(* Logix 5000 project; controller Lift_Station_Template vendor 1 type 14 code 196 rev 32.11; software revision 32.00 *)

TASK MainTask (continuous, watchdog 500 ms) : InLink, MainProgram, OutLink

MODULES
   Local : vendor 1 type 14 code 196 (5069 0, rev 32.11)
      DI_01 : 5069-IB16 (5069 1, rev 2.1, StandardDataDriven RPI 5 ms)
      DO_02 : 5069-OB16 (5069 2, rev 2.1, StandardDataDriven RPI 5 ms)
END_MODULES

TYPE Pump :
STRUCT
   HOA_Auto : BOOL;   // Physical HOA in Auto
   ManStartPB : BOOL;
   ManStopPB : BOOL;
   AutoStart : BOOL;
   CallToRun : BOOL;
   Running : BOOL;
   FailToRun : DiscreteAlarm;
   StartCount : DINT;
   ManSS : BOOL;
END_STRUCT
END_TYPE

ADD_ON_INSTRUCTION DiscreteAlarm   (* revision 1.0 *)
VAR_INPUT
   Trigger : BOOL; {required}
   Delay : DINT; {required}
   Supress : BOOL; {visible}
   Disable : BOOL; {visible}
END_VAR
VAR_OUTPUT
   Alarm : BOOL; {required}
   Acc : DINT; {visible}
END_VAR
VAR_INPUT
   Latching : BOOL; {visible}
   Reset : BOOL;
END_VAR
VAR
   DelayTmr : TIMER; {access None}
END_VAR

ROUTINE Logic   (* ladder *)
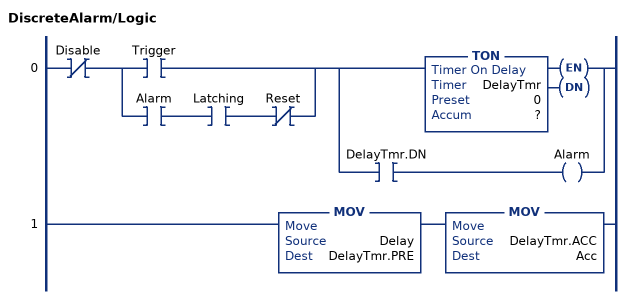
   0: XIO(Disable)[XIC(Trigger) ,XIC(Alarm) XIC(Latching) XIO(Reset) ][TON(DelayTmr,?,?) ,XIC(DelayTmr.DN) OTE(Alarm) ];
   1: MOV(Delay,DelayTmr.PRE)MOV(DelayTmr.ACC,Acc);
END_ROUTINE
END_ADD_ON_INSTRUCTION

VAR_GLOBAL   (* controller tags *)
   LSH_2 : BOOL;
   LSL_1 : BOOL;
   ONS : DINT[5];
   Pump : Pump[4];
   PumpReqCount : DINT;
   PumpRequired : BOOL;
   StageUpTmr : TIMER := (PRE := 300000);
END_VAR

PROGRAM InLink   (* main routine _00_Main *)
// Input Linking

ROUTINE _00_Main   (* ladder *)
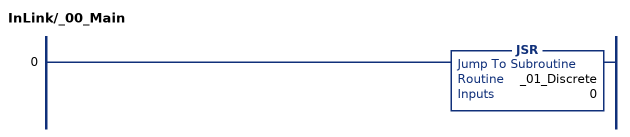
   0: JSR(_01_Discrete,0);
END_ROUTINE

ROUTINE _01_Discrete   (* ladder *)
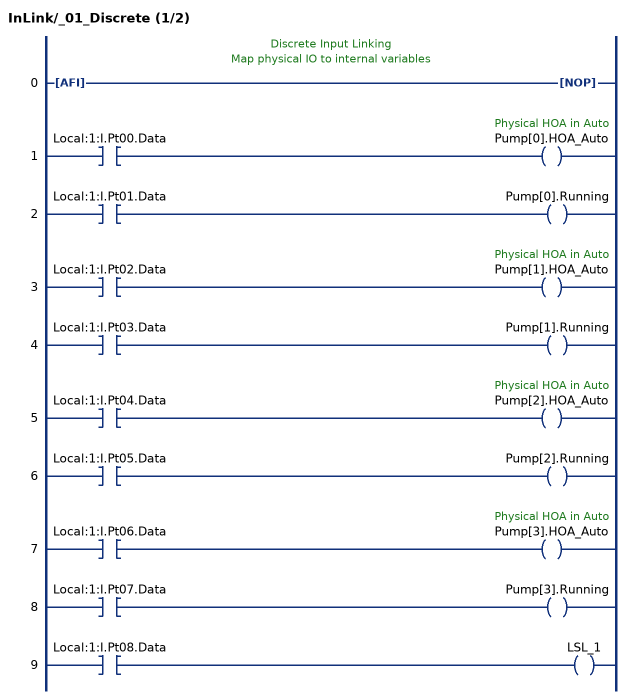
   // Discrete Input Linking
   // Map physical IO to internal variables
   0: AFI()NOP();
   1: XIC(Local:1:I.Pt00.Data)OTE(Pump[0].HOA_Auto);
   2: XIC(Local:1:I.Pt01.Data)OTE(Pump[0].Running);
   3: XIC(Local:1:I.Pt02.Data)OTE(Pump[1].HOA_Auto);
   4: XIC(Local:1:I.Pt03.Data)OTE(Pump[1].Running);
   5: XIC(Local:1:I.Pt04.Data)OTE(Pump[2].HOA_Auto);
   6: XIC(Local:1:I.Pt05.Data)OTE(Pump[2].Running);
   7: XIC(Local:1:I.Pt06.Data)OTE(Pump[3].HOA_Auto);
   8: XIC(Local:1:I.Pt07.Data)OTE(Pump[3].Running);
   9: XIC(Local:1:I.Pt08.Data)OTE(LSL_1);
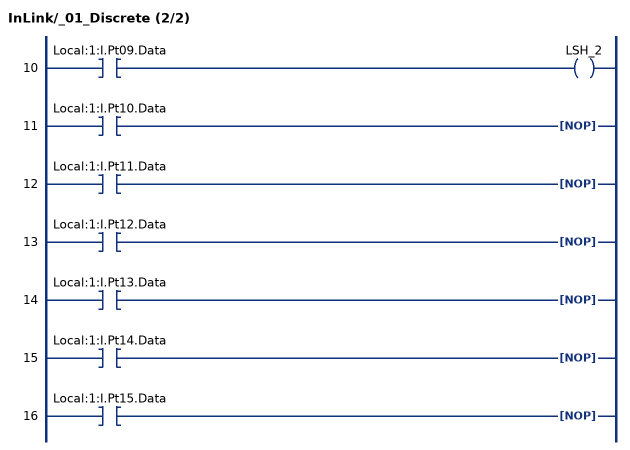
   10: XIC(Local:1:I.Pt09.Data)OTE(LSH_2);
   11: XIC(Local:1:I.Pt10.Data)NOP();
   12: XIC(Local:1:I.Pt11.Data)NOP();
   13: XIC(Local:1:I.Pt12.Data)NOP();
   14: XIC(Local:1:I.Pt13.Data)NOP();
   15: XIC(Local:1:I.Pt14.Data)NOP();
   16: XIC(Local:1:I.Pt15.Data)NOP();
END_ROUTINE
END_PROGRAM

PROGRAM MainProgram   (* main routine _00_MainRoutine *)

ROUTINE _00_MainRoutine   (* ladder *)
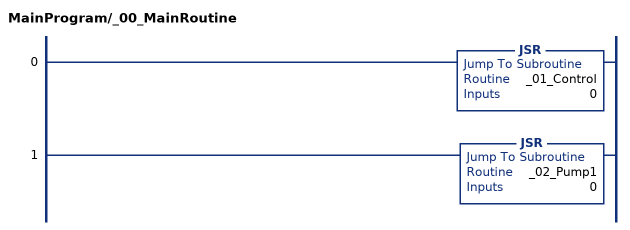
   0: JSR(_01_Control,0);
   1: JSR(_02_Pump1,0);
END_ROUTINE

ROUTINE _01_Control   (* ladder *)
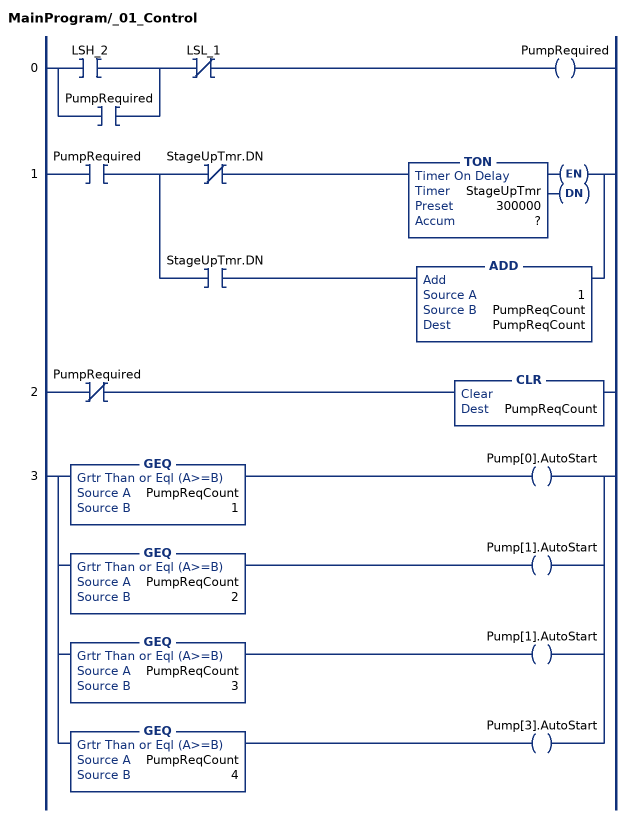
   0: [XIC(LSH_2) ,XIC(PumpRequired) ]XIO(LSL_1)OTE(PumpRequired);
   1: XIC(PumpRequired)[XIO(StageUpTmr.DN) TON(StageUpTmr,?,?) ,XIC(StageUpTmr.DN) ADD(1,PumpReqCount,PumpReqCount) ];
   2: XIO(PumpRequired)CLR(PumpReqCount);
   3: [GEQ(PumpReqCount,1) OTE(Pump[0].AutoStart) ,GEQ(PumpReqCount,2) OTE(Pump[1].AutoStart) ,GEQ(PumpReqCount,3) OTE(Pump[1].AutoStart) ,GEQ(PumpReqCount,4) OTE(Pump[3].AutoStart) ];
END_ROUTINE

ROUTINE _02_Pump1   (* ladder *)
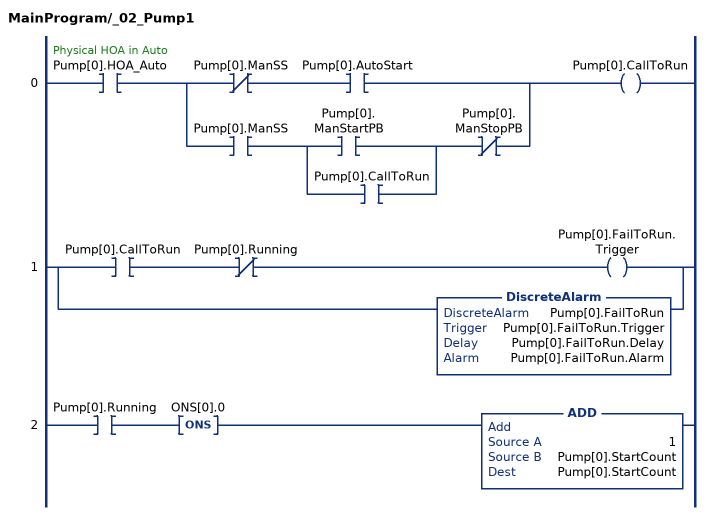
   0: XIC(Pump[0].HOA_Auto)[XIO(Pump[0].ManSS) XIC(Pump[0].AutoStart) ,XIC(Pump[0].ManSS) [XIC(Pump[0].ManStartPB) ,XIC(Pump[0].CallToRun) ] XIO(Pump[0].ManStopPB) ]OTE(Pump[0].CallToRun);
   1: [XIC(Pump[0].CallToRun) XIO(Pump[0].Running) OTE(Pump[0].FailToRun.Trigger) ,DiscreteAlarm(Pump[0].FailToRun,Pump[0].FailToRun.Trigger,Pump[0].FailToRun.Delay,Pump[0].FailToRun.Alarm) ];
   2: XIC(Pump[0].Running)ONS(ONS[0].0)ADD(1,Pump[0].StartCount,Pump[0].StartCount);
END_ROUTINE

ROUTINE _03_Pump2   (* ladder *)
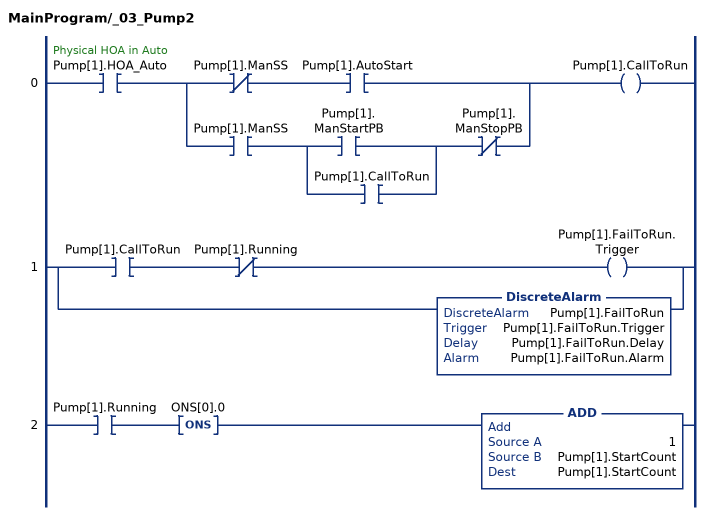
   0: XIC(Pump[1].HOA_Auto)[XIO(Pump[1].ManSS) XIC(Pump[1].AutoStart) ,XIC(Pump[1].ManSS) [XIC(Pump[1].ManStartPB) ,XIC(Pump[1].CallToRun) ] XIO(Pump[1].ManStopPB) ]OTE(Pump[1].CallToRun);
   1: [XIC(Pump[1].CallToRun) XIO(Pump[1].Running) OTE(Pump[1].FailToRun.Trigger) ,DiscreteAlarm(Pump[1].FailToRun,Pump[1].FailToRun.Trigger,Pump[1].FailToRun.Delay,Pump[1].FailToRun.Alarm) ];
   2: XIC(Pump[1].Running)ONS(ONS[0].0)ADD(1,Pump[1].StartCount,Pump[1].StartCount);
END_ROUTINE

ROUTINE _04_Pump3   (* ladder *)
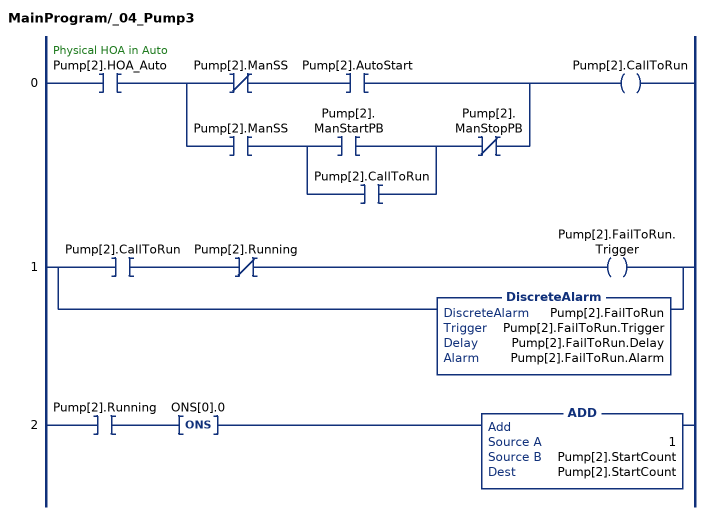
   0: XIC(Pump[2].HOA_Auto)[XIO(Pump[2].ManSS) XIC(Pump[2].AutoStart) ,XIC(Pump[2].ManSS) [XIC(Pump[2].ManStartPB) ,XIC(Pump[2].CallToRun) ] XIO(Pump[2].ManStopPB) ]OTE(Pump[2].CallToRun);
   1: [XIC(Pump[2].CallToRun) XIO(Pump[2].Running) OTE(Pump[2].FailToRun.Trigger) ,DiscreteAlarm(Pump[2].FailToRun,Pump[2].FailToRun.Trigger,Pump[2].FailToRun.Delay,Pump[2].FailToRun.Alarm) ];
   2: XIC(Pump[2].Running)ONS(ONS[0].0)ADD(1,Pump[2].StartCount,Pump[2].StartCount);
END_ROUTINE

ROUTINE _05_Pump4   (* ladder *)
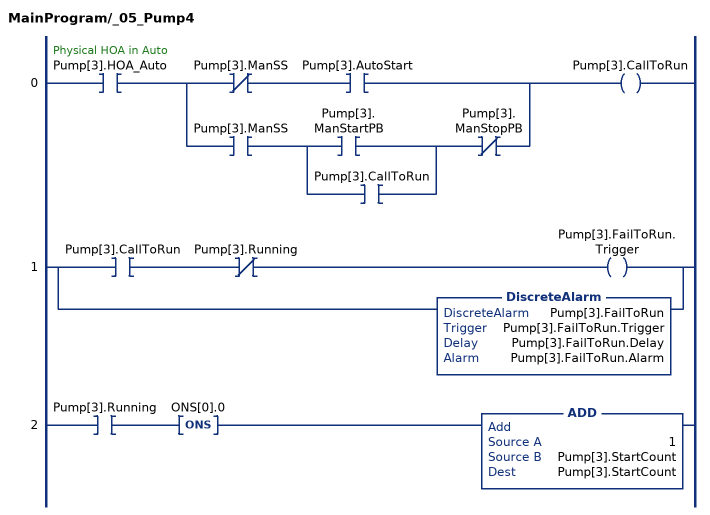
   0: XIC(Pump[3].HOA_Auto)[XIO(Pump[3].ManSS) XIC(Pump[3].AutoStart) ,XIC(Pump[3].ManSS) [XIC(Pump[3].ManStartPB) ,XIC(Pump[3].CallToRun) ] XIO(Pump[3].ManStopPB) ]OTE(Pump[3].CallToRun);
   1: [XIC(Pump[3].CallToRun) XIO(Pump[3].Running) OTE(Pump[3].FailToRun.Trigger) ,DiscreteAlarm(Pump[3].FailToRun,Pump[3].FailToRun.Trigger,Pump[3].FailToRun.Delay,Pump[3].FailToRun.Alarm) ];
   2: XIC(Pump[3].Running)ONS(ONS[0].0)ADD(1,Pump[3].StartCount,Pump[3].StartCount);
END_ROUTINE
END_PROGRAM

PROGRAM OutLink   (* main routine _00_Main *)

ROUTINE _00_Main   (* ladder *)
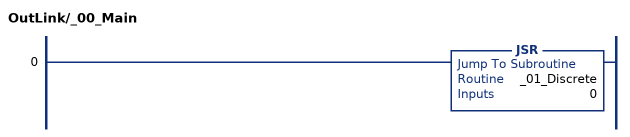
   0: JSR(_01_Discrete,0);
END_ROUTINE

ROUTINE _01_Discrete   (* ladder *)
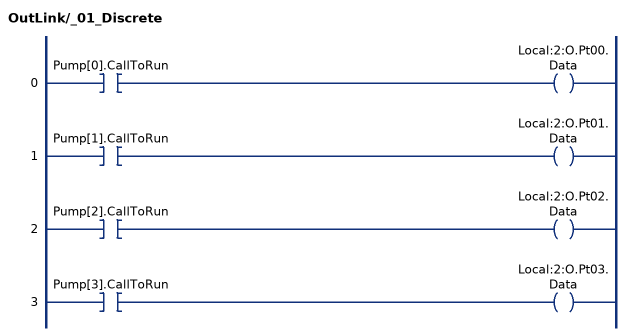
   0: XIC(Pump[0].CallToRun)OTE(Local:2:O.Pt00.Data);
   1: XIC(Pump[1].CallToRun)OTE(Local:2:O.Pt01.Data);
   2: XIC(Pump[2].CallToRun)OTE(Local:2:O.Pt02.Data);
   3: XIC(Pump[3].CallToRun)OTE(Local:2:O.Pt03.Data);
END_ROUTINE
END_PROGRAM
